{attribute 'GeneratedUsingTerminal: EL6001-0000-0020'}
{attribute addProperty BoxType "EL6001-0000-0020"}
{attribute addProperty Id "CtrlAT %Q*Ctrl_71604E865Data_OutAT %Q*ARRAY[0..21] OF USINT22"}
{attribute addProperty CRC "2695605661"}
{attribute addProperty Size "27"}
TYPE COM_Outputs_DEF408EC EXTENDS TcoIo.OutputBase_10CEE7DE :
STRUCT
	{attribute addProperty Name "Ctrl"}
	Ctrl AT %Q* : Ctrl_71604E86;
	{attribute addProperty Name "Data_Out"}
	Data_Out AT %Q* : ARRAY[0..21] OF USINT;
END_STRUCT
END_TYPE

(* stored: Version 1.2.0.0, ProductVersion 3.1.4024.11
   DUT COM_Outputs_DEF408EC: Id {6cd4de5e-4aa4-44d5-b8f7-3e2970dff412} *)
